// TwinCAT 3 PLC project UnitTests
// ProgramVersion: 3.1.4023.0
// libraries:
//   Tc2_Standard, * (Beckhoff Automation GmbH)
//   Tc2_System, * (Beckhoff Automation GmbH)
//   Tc2_Utilities, * (Beckhoff Automation GmbH)
//   Tc3_Module, * (Beckhoff Automation GmbH)
//   TcUnit, * (www.tcunit.org)
// project tree:
//   DUTs/ ST_BoolHmi.TcDUT
//   General/ E_OpMode.TcDUT, FB_Unit.TcPOU
//   GVLs/ IO.TcGVL
//   / PlcTask.TcTTO, POU_Test.TcPOU
//   POUs/ MAIN.TcPOU
//   RotaryMovement/ E_Direction.TcDUT, FB_SewMovitracBFieldbus.TcPOU, FB_SimpleRotaryTwoWayDrive.TcPOU, ST_SewControlWord.TcDUT, ST_SewStatusWord.TcDUT, ST_SimpleRotaryTwoWayDriveControl.TcDUT, ST_SimpleRotaryTwoWayDriveStatus.TcDUT, U_SewControlWord1.TcDUT, U_SewStatusWord1.TcDUT
//   RotaryMovement/Test/ FB_SewMovitracBFieldbusTest.TcPOU
//   TwoPointMovement/ FB_LinearMovementWithFeedback.TcPOU, FB_SimpleLinearTwoWayDrive.TcPOU, ST_SimpleLinearTwoWayDriveHmi.TcDUT
//   TwoPointMovement/Test/ FB_LinearMovementWithFeedbackTest.TcPOU, FB_SimpleLinearTwoWayDrive_Test.TcPOU
// real-time tasks:
//   TASK PlcTask: cycle T#10ms, priority 20, ADS port 350

CONFIGURATION UnitTests
    RESOURCE PLC ON TwinCAT3
        TASK PlcTask(INTERVAL := T#10ms, PRIORITY := 20);
        PROGRAM MAIN WITH PlcTask : MAIN;
        PROGRAM POU_Test WITH PlcTask : POU_Test;
    END_RESOURCE
END_CONFIGURATION

// ---- DUTs/ST_BoolHmi.TcDUT
TYPE ST_BoolHmi :
STRUCT
	Enabled: BOOL;
	PlcToHmi: BOOL;
	HmiToPlc: BOOL;
END_STRUCT
END_TYPE

// ---- General/E_OpMode.TcDUT
{attribute 'qualified_only'}
{attribute 'strict'}
TYPE E_OpMode :
(
	Stop,
	Manual, 
	Jog,
	Automatic,
	AutomaticRunning
);
END_TYPE

// ---- RotaryMovement/E_Direction.TcDUT
{attribute 'qualified_only'}
{attribute 'strict'}
TYPE E_Direction :
(
	Right_Forward_Up,
	Left_Back_Down
);
END_TYPE

// ---- RotaryMovement/ST_SewControlWord.TcDUT
TYPE ST_SewControlWord :
STRUCT
	ControllerInhibit:			BIT; 	// (bit 0) inhibit="1", enable="0"
	EnableElseRapidStop:		BIT;	// (bit 1) enable=1", rapid stop="0"
	EnableElseStop:				BIT;	// (bit 2) enable="1", stop="0"
	HoldControl:				BIT;	// (bit 3) not relevant
	IntegratorSwitchover:		BIT;	// (bit 4) not relevant
	ParameterSetSwitchOver:		BIT;	// (bit 5) not relevant
	Reset:						BIT;	// (bit 6) reset="1"
	Reserved1:					BIT;	// (bit 7) set reserved bits to zero
	DirectionOfRotation:		BIT;	// (bit 8) 0=CW direction of rotation, 1=CCW direction of rotation
	AccelerationDecceleration1: BIT;	// (bit 9) Works together with next bit
	AccelerationDecceleration2:	BIT;	// (bit 10) 00=no change, 01=down, 10=up, 11=no change
	FixedSetpoints1:			BIT;	// (bit 11) works together with next bit
	FixedSetpoints2:			BIT;	// (bit 12) 00=speed setpoint via process output data word 2, 10=internal setpoint n11, 01=internal setpoint n12, 11=internal setpoint n13
	FixedSetpointSwitchover:	BIT;	// (bit 13) 0=fixed setpoints of the active parameter set selectable via bit 11/22, 1=fixed setpoint of the other parameter set selectable via bit 11/12
	Reserved2:					BIT;	// (bit 14) set reserved bits to zero
	Reserved3:					BIT;	// (bit 15) set reserved bits to zero
END_STRUCT
END_TYPE

// ---- RotaryMovement/ST_SewStatusWord.TcDUT
TYPE ST_SewStatusWord :
STRUCT
	OutputStageEnabled: 		BIT;	// enabled="1", inhibited="0"
	InverterReady: 				BIT;	// ready="1", not ready="0"
	PODataEnabled: 				BIT;	// enabled="1", disabled="0"
	CurrentRampGEneratorSet: 	BIT;	// Integrator 2="1", Integrator 1="0"
	CurrentParameterSet: 		BIT;	// Parameter set 2="1", Parameter set 1="0"
	FaultOrWarning:				BIT;	// pending="1", no fault="0"
	CWLimitSwitchActive:		BIT;	// active="1", inactive="0"
	CCWLimitSwitchACtive:		BIT;	// active="1", inactive="0"
END_STRUCT
END_TYPE

// ---- RotaryMovement/ST_SimpleRotaryTwoWayDriveControl.TcDUT
TYPE ST_SimpleRotaryTwoWayDriveControl :
STRUCT
	Enable: 	BOOL;
	Lock:		BOOL;
	Run: 		BOOL;
	Reset:		BOOL;
	Speed:		UINT; 
	Direction: 	E_Direction;
END_STRUCT
END_TYPE

// ---- RotaryMovement/ST_SimpleRotaryTwoWayDriveStatus.TcDUT
TYPE ST_SimpleRotaryTwoWayDriveStatus :
STRUCT
	Ready: 	BOOL; 			(* Inverter is ready for operation *)
	Warning: BOOL; 			(* Inverter is in warning state *)
	Malfunction: BOOL; 		(* Inverter malfunctions *)
	Speed: REAL; 			(* Speed 0-100% *)
	OutputCurrent: REAL; 	(* output current in [A] *)
END_STRUCT
END_TYPE

// ---- RotaryMovement/U_SewControlWord1.TcDUT
TYPE U_SewControlWord1 :
UNION
	nUINT:	UINT;
	aBits:	ST_SewControlWord;
END_UNION
END_TYPE

// ---- RotaryMovement/U_SewStatusWord1.TcDUT
TYPE U_SewStatusWord1 :
UNION
	nUint: UINT;
	aBits: ST_SewSTatusWord;
END_UNION
END_TYPE

// ---- TwoPointMovement/ST_SimpleLinearTwoWayDriveHmi.TcDUT
TYPE ST_SimpleLinearTwoWayDriveHmi :
STRUCT
	 ToHomePos: ST_BoolHmi;
	 ToWorkPos: ST_BoolHmi;
END_STRUCT
END_TYPE

// ---- GVLs/IO.TcGVL
{attribute 'qualified_only'}
VAR_GLOBAL
	OP1_A100 AT %I*: BOOL; 
END_VAR

// ---- POUs/MAIN.TcPOU
PROGRAM MAIN
VAR
END_VAR

END_PROGRAM

// ---- POU_Test.TcPOU
PROGRAM POU_Test
VAR
	fbSimpleLinearTwoWayDriveTest: FB_SimpleLinearTwoWayDrive_Test; 
	fbLinearMovementWithFeedbackTest: FB_LinearMovementWithFeedbackTest;
	fbSewMovitracBFieldbusTest: FB_SewMovitracBFieldbusTest;
END_VAR

TcUnit.RUN();

END_PROGRAM

// ---- TwoPointMovement/Test/FB_SimpleLinearTwoWayDrive_Test.TcPOU
FUNCTION_BLOCK FB_SimpleLinearTwoWayDrive_Test EXTENDS FB_TestSuite
VAR_INPUT
END_VAR
VAR_OUTPUT
END_VAR

Trigger_movement_from_hmi();

METHOD Trigger_movement_from_code : BOOL
VAR_INPUT
END_VAR
VAR
	sut: FB_SimpleLinearTwoWayDrive;
	result : BOOL := TRUE;
	
	Hmi : ST_SimpleLinearTwoWayDriveHmi;
END_VAR
TEST('Movement executes when triggered from code');

Hmi.ToHomePos.HmiToPlc := FALSE;

sut(
	OpMode := E_OpMode.AutomaticRunning,
	SensorHomePos := FALSE,
	ToHome := TRUE,
	Enable := TRUE,
	Hmi := Hmi);
	
AssertEquals(result, sut.ActorHomePos, 'Movement does not start');

TEST_FINISHED();
END_METHOD

METHOD Trigger_movement_from_hmi : BOOL
VAR_INPUT
END_VAR
VAR
	sut: FB_SimpleLinearTwoWayDrive;
	result : BOOL := TRUE;
	
	Hmi : ST_SimpleLinearTwoWayDriveHmi;
END_VAR
TEST('Movement executes when triggered from HMI');

Hmi.ToHomePos.HmiToPlc := TRUE;

sut(
	OpMode := E_OpMode.Manual,
	SensorHomePos := FALSE,
	Enable := TRUE,
	Hmi := Hmi);
	
AssertEquals(result, sut.ActorHomePos, 'Movement does not start');

TEST_FINISHED();
END_METHOD

END_FUNCTION_BLOCK

// ---- TwoPointMovement/FB_SimpleLinearTwoWayDrive.TcPOU
FUNCTION_BLOCK FB_SimpleLinearTwoWayDrive EXTENDS FB_Unit
VAR_INPUT
	SensorHomePos: BOOL;
	SensorWorkPos: BOOL;
	Enable: BOOL;
	LockHomePos: BOOL;
	LockWorkPos: BOOL;
	HoldPosition: BOOL;	// TRUE: Hold output to true even if position has been reached
	ToHome: BOOL;
	ToWork: BOOL;
END_VAR
VAR_OUTPUT	
	ActorHomePos: BOOL;
	ActorWorkPos: BOOL;
END_VAR
VAR
	toHomePos: BOOL;
	toWorkPos: BOOL;
	HomePos: FB_LinearMovementWithFeedback;
	WorkPos: FB_LinearMovementWithFeedback;
END_VAR
VAR_IN_OUT
	Hmi: ST_SimpleLinearTwoWayDriveHmi;
END_VAR

// This could be refactored further by adding a data structure instead of inputs.
// advantages:
// - could be transferred to HMI
// - further removal of code dublication
// disadvantages:
// - adds another layer of indirection, e.g. for cross-reference search

toHomePos :=
	(SUPER^.OpMode = E_OpMode.Manual AND Hmi.ToHomePos.HmiToPlc)
	OR
	(SUPER^.OpMode = E_OpMode.Automatic AND ToHome);
	
toWorkPos :=
	(SUPER^.OpMode = E_OpMode.Manual AND Hmi.ToWorkPos.HmiToPlc)
	OR
	(SUPER^.OpMode = E_OpMode.Automatic AND ToHome);

HomePos(
	ToPosition := toHomePos,
	Feedback := SensorHomePos,
	Lock := NOT Enable OR LockHomePos OR toWorkPos,
	HoldOutput := HoldPosition,
	Actor => ActorHomePos);
	
WorkPos(
	ToPosition := toWorkPos,
	Feedback := SensorWorkPos,
	Lock := NOT Enable OR LockWorkPos OR toHomePos,
	HoldOutput := HoldPosition,
	Actor => ActorWorkPos);

END_FUNCTION_BLOCK

// ---- General/FB_Unit.TcPOU
FUNCTION_BLOCK FB_Unit
VAR_INPUT
	OpMode: E_OpMode;
END_VAR
VAR_OUTPUT
END_VAR
VAR
END_VAR

END_FUNCTION_BLOCK

// ---- TwoPointMovement/FB_LinearMovementWithFeedback.TcPOU
FUNCTION_BLOCK FB_LinearMovementWithFeedback
VAR_INPUT
	ToPosition: BOOL;	// TRUE: Moves the drive to position
	Feedback:	BOOL;	// Feedback signal (e.g. reed contact)
	Lock: 		BOOL;	// Interlock for the output
	HoldOutput: BOOL;	// TRUE: Actor remains true when target position reached
END_VAR
VAR_OUTPUT
	Actor:		BOOL;	
END_VAR
VAR
END_VAR

Actor := ToPosition AND NOT Lock AND (HoldOutput OR NOT Feedback);

END_FUNCTION_BLOCK

// ---- TwoPointMovement/Test/FB_LinearMovementWithFeedbackTest.TcPOU
FUNCTION_BLOCK FB_LinearMovementWithFeedbackTest EXTENDS FB_TestSuite
VAR_INPUT
END_VAR
VAR_OUTPUT
END_VAR
VAR
END_VAR

Movement_stops_when_position_is_reached();
Movement_executes_when_triggered();
Output_is_still_active_when_position_has_been_reached_but_holdPos_has_been_set();
No_Movement_When_Direction_Is_Locked();

METHOD Movement_executes_when_triggered : BOOL
VAR_INPUT
END_VAR
VAR
	sut: FB_LinearMovementWithFeedback;
	result : BOOL := TRUE;
END_VAR
TEST('Movement executes when triggered');

sut(
	ToPosition:= TRUE,
	Feedback:= FALSE,
	Lock:= FALSE,
	HoldOutput:= FALSE);
	
AssertEquals(result, sut.Actor, 'Movement does not start');

TEST_FINISHED();
END_METHOD

METHOD Movement_stops_when_position_is_reached : BOOL
VAR_INPUT
END_VAR
VAR_INST
	sut: FB_LinearMovementWithFeedback;
	result : BOOL := FALSE;
END_VAR
TEST('Movement stops when position is reached');

sut(
	ToPosition:= TRUE,
	Feedback:= True,
	Lock:= FALSE,
	HoldOutput:= FALSE);
	
AssertEquals(result, sut.Actor, 'Movement even if not enabled');

TEST_FINISHED();
END_METHOD

METHOD No_Movement_When_Direction_Is_Locked : BOOL
VAR_INPUT
END_VAR
VAR
	sut: FB_LinearMovementWithFeedback;
	result : BOOL := FALSE;
END_VAR
TEST('Output should remain set when position is reached but Hold is set');

sut(
	ToPosition:= TRUE,
	Feedback:= FALSE,
	Lock:= TRUE,
	HoldOutput:= FALSE);
	
AssertEquals(result, sut.Actor, 'Target reached but output not hold.');

TEST_FINISHED();
END_METHOD

METHOD Output_is_still_active_when_position_has_been_reached_but_holdPos_has_been_set : BOOL
VAR_INPUT
END_VAR
VAR
	sut: FB_LinearMovementWithFeedback;
	result : BOOL := TRUE;
END_VAR
TEST('Output remains set when position has been reached when setting hold pos is true');

sut(
	ToPosition:= TRUE,
	Feedback:= True,
	Lock:= FALSE,
	HoldOutput:= TRUE);
	
AssertEquals(result, sut.Actor, '');

TEST_FINISHED();
END_METHOD

END_FUNCTION_BLOCK

// ---- RotaryMovement/Test/FB_SewMovitracBFieldbusTest.TcPOU
FUNCTION_BLOCK FB_SewMovitracBFieldbusTest EXTENDS FB_TestSuite
VAR_INPUT
END_VAR
VAR_OUTPUT
END_VAR
VAR
END_VAR

StartDrive();
HaltDrive();
RunWithSetSpeed();
ReadWarning();

METHOD HaltDrive : BOOL
VAR
	sut: FB_SewMovitracBFieldbus;
	control : ST_SimpleRotaryTwoWayDriveControl;
	result : UINT := 2#0000_1111_0000_0000; // SEW: Big Endian, TwinCAT: Little Endian
END_VAR
TEST('Halt drive');

control.Enable := TRUE;
control.Lock := TRUE;

sut(
	PI1 := 0,
	PI2 := 0,
	PI3 := 0,
	Control := control);
	
AssertEquals(result, sut.PO1.nUINT, 'Drive does not halt');

TEST_FINISHED();
END_METHOD

METHOD ReadWarning : BOOL
VAR_INPUT
END_VAR
VAR
	sut: FB_SewMovitracBFieldbus;
	result : BOOL := TRUE; 
END_VAR
TEST('Read warning');

sut(
	PI1 := 2#0010_0010_0000_0000,
	PI2 := 0,
	PI3 := 0);
	
AssertEquals(result, sut.Status.Warning, 'Warning not correctly decoded.');

TEST_FINISHED();
END_METHOD

METHOD RunWithSetSpeed : BOOL
VAR_INPUT
END_VAR
VAR
	sut: FB_SewMovitracBFieldbus;
	control : ST_SimpleRotaryTwoWayDriveControl;
	result : UINT := 2#0000_0110_0000_0000; // SEW: Big Endian, TwinCAT: Little Endian 
	resultSpeed : UINT := HOST_TO_BE16(80);
END_VAR
TEST('Run with set speed');

control.Direction := E_Direction.Right_Forward_Up;
control.Enable := TRUE;
control.Run := TRUE;
control.Speed := 80;

sut(
	PI1 := 0,
	PI2 := 0,
	PI3 := 0, 
	Control := control);

AssertEquals(result, sut.PO1.nUINT, 'Drive does not run with set speed');
AssertEquals(resultSpeed, sut.PO2, 'Drive does not run with set speed');

TEST_FINISHED();
END_METHOD

METHOD StartDrive : BOOL
VAR
	sut: FB_SewMovitracBFieldbus;
	control : ST_SimpleRotaryTwoWayDriveControl;
	result : UINT := 2#0000_0110_0000_0000; // SEW: Big Endian, TwinCAT: Little Endian
END_VAR
TEST('Start drive');

control.Direction := E_Direction.Right_Forward_Up;
control.Enable := TRUE;
control.Run := TRUE;

sut(
	PI1 := 0,
	PI2 := 0,
	PI3 := 0,
	Control := control);
	
AssertEquals(result, sut.PO1.nUINT, 'Drive does not start');

TEST_FINISHED();
END_METHOD

END_FUNCTION_BLOCK

// ---- RotaryMovement/FB_SewMovitracBFieldbus.TcPOU
FUNCTION_BLOCK FB_SewMovitracBFieldbus
VAR_INPUT
	PI1: UINT;	(* Process input data 1: status word *)
	PI2: UINT;	(* Process input data 2: speed *)
	PI3: UINT;	(* Process input data 3: output current *)
	Control: ST_SimpleRotaryTwoWayDriveControl;
END_VAR
VAR_OUTPUT
	PO1: U_SewControlWord1;	(* Process output data 1: control word *)
	PO2: UINT;	(* Process output data 2: speed *)
	PO3: UINT;	(* Process output data 3: not used *)
	Status: ST_SimpleRotaryTwoWayDriveStatus; 
END_VAR
VAR
	StatusWord1: U_SewStatusWord1;
END_VAR

// Set outputs
PO1 := SetPO1();
PO2 := HOST_TO_BE16(LIMIT(0, Control.Speed, 100));
PO3 := 0;

// Process inputs
StatusWord1.nUint := BE16_TO_HOST(in:=PI1);

Status.Warning := StatusWord1.aBits.InverterReady AND StatusWord1.aBits.FaultOrWarning;
Status.Ready := StatusWord1.aBits.InverterReady AND NOT StatusWord1.aBits.FaultOrWarning;
Status.Malfunction := NOT StatusWord1.aBits.InverterReady AND StatusWord1.aBits.FaultOrWarning;
Status.Speed := BE16_TO_HOST(in:=PI2);
Status.OutputCurrent := BE16_TO_HOST(in:=PI3);

METHOD PRIVATE SetPO1 : U_SewControlWord1
VAR_INPUT
END_VAR
VAR
	PO1_LittleEndian: U_SewControlWord1;
END_VAR
// Bit 0: Controller inhibit
PO1_LittleEndian.aBits.ControllerInhibit := Control.Lock;
// Bit 1 & 2: Enable
PO1_LittleEndian.aBits.EnableElseRapidStop := Control.Enable;
PO1_LittleEndian.aBits.EnableElseStop := Control.Enable;
// Bit 3: Hold Control
PO1_LittleEndian.aBits.HoldControl := NOT Control.Run;
// Bit 4 & 5: not used
PO1_LittleEndian.aBits.IntegratorSwitchover := FALSE;
PO1_LittleEndian.aBits.ParameterSetSwitchOver := FALSE;
// Bit 6: Reset
PO1_LittleEndian.aBits.Reset := Control.Reset;
// Bit 7: Reserved
PO1_LittleEndian.aBits.Reserved1 := FALSE;
// Bit 8: Direction of rotation
IF Control.Direction = E_Direction.Right_Forward_Up THEN
	PO1_LittleEndian.aBits.DirectionOfRotation := FALSE;
ELSE
	PO1_LittleEndian.aBits.DirectionOfRotation := TRUE;
END_IF
// Bit 9 & 10: Acc / Decc => not used
PO1_LittleEndian.aBits.AccelerationDecceleration1 := FALSE;
PO1_LittleEndian.aBits.AccelerationDecceleration2 := FALSE;
// Bit 11 & 12: Selection of internal fixed setpoint => set to use setpoint via PO2
PO1_LittleEndian.aBits.FixedSetpoints1 := FALSE;
PO1_LittleEndian.aBits.FixedSetpoints2 := FALSE;
// Bit 13: Fixed setpoint switch over => not used
PO1_LittleEndian.aBits.FixedSetpointSwitchover := FALSE;
// Bit 14 & 15: reserved
PO1_LittleEndian.aBits.Reserved2 := FALSE;
PO1_LittleEndian.aBits.Reserved3 := FALSE;

// Convert to Big Endian
SetPO1.nUINT := HOST_TO_BE16(in := PO1_LittleEndian.nUINT);
END_METHOD

END_FUNCTION_BLOCK

// ---- RotaryMovement/FB_SimpleRotaryTwoWayDrive.TcPOU
FUNCTION_BLOCK FB_SimpleRotaryTwoWayDrive EXTENDS FB_Unit
VAR_INPUT
END_VAR
VAR_OUTPUT
END_VAR
VAR
END_VAR

END_FUNCTION_BLOCK
